{attribute 'qualified_only'}
{attribute 'strict'}
{attribute 'to_string'}
TYPE DataTrigger :
(
	none	:= 0,
	x		:= 1,
	y		:= 2,
	z		:= 3,
	time1	:= 4
);
END_TYPE

(* stored: Version 1.1.0.1, ProductVersion 3.1.4026.12
   DUT DataTrigger: Id {be471f01-f0e0-445d-b6e1-ee3726564ad3} *)
